FUNCTION_BLOCK FB_TcEvent
VAR_INPUT
	sName							:STRING;
	stPosData						:ST_PosData;
	bAck							:BOOL;
	stEventEntry					:TcEventEntry;				(*Event definition*)
	aErrorDesc					:ARRAY [0..31] OF STRING;
END_VAR
VAR_OUTPUT
	sError						:STRING(255);					(*hiba string*)
END_VAR
VAR
	i							:INT;
	nErrorCodeTmp				:UDINT;
	bIsInitalized				:BOOL;
	fbAlarm						:FB_TcAlarm;
	fbErrorRTrig				:R_Trig;
	fbAckRTrig					:R_Trig;
END_VAR

IF stPosData.bError THEN
	sError := sName;
	nErrorCodeTmp :=  stPosData.nErrorCode;
	FOR i:=0 TO 31 DO
		IF nErrorCodeTmp.0 THEN
			sError :=  CONCAT(sError, aErrorDesc[i]);
		END_IF
		nErrorCodeTmp := SHR(nErrorCodeTmp,1);
	END_FOR
ELSE
	sError := '';
END_IF

(*Hiba kezelés Tc3_EventLogger*)
IF NOT bIsInitalized THEN
	bIsInitalized := TRUE;
	fbAlarm.CreateEx(stEventEntry, TRUE, 0);
END_IF

fbErrorRTrig(CLK:= stPosData.bError);
fbAckRTrig(CLK:= bAck);

(*Hiba generálás*)
IF fbErrorRTrig.Q THEN
	fbAlarm.ipArguments.Clear().AddString(sError);
	fbAlarm.Raise(0);
END_IF
(*Hiba nyugtázás*)
IF fbAckRTrig.Q THEN
	fbAlarm.Confirm(0);
END_IF
(*Hiba törlés (nyugtázott és megszűnt)*)
IF fbAlarm.eConfirmationState = 3 AND NOT stPosData.bError THEN
	fbAlarm.Clear(0, FALSE);
END_IF

END_FUNCTION_BLOCK

(* stored: Version 1.1.0.1, ProductVersion 3.1.4024.11
   POU FB_TcEvent: Id {b22169a4-b9e3-4549-a1f5-1ec0749d241c}, SpecialFunc None *)
